FUNCTION_BLOCK FB_LensCompounderMock EXTENDS FB_FallibleMock IMPLEMENTS I_LensCompounder
VAR
    fFocalLengthCompounded : LREAL;
END_VAR


METHOD Compound : LREAL
VAR_INPUT
    fFocalLength	: LREAL;
    nMultiplier	: INT;
END_VAR
END_METHOD


PROPERTY FocalLengthCompounded : LREAL
GET

FocalLengthCompounded := fFocalLengthCompounded;
END_GET
SET

fFocalLengthCompounded := FocalLengthCompounded;
END_SET
END_PROPERTY


METHOD Reset
END_METHOD


METHOD SetValid

FocalLengthCompounded := 1.0;
ClearError();
END_METHOD

END_FUNCTION_BLOCK

(* stored: Version 1.1.0.1
   POU FB_LensCompounderMock: Id {f3a1ef28-98f7-4a8c-a126-ddef21ffe39c}, SpecialFunc None
   Method Compound: Id {785c0eab-8b59-435e-bd8e-fdfd5fe072fc}
   Property FocalLengthCompounded: Id {6ab06aab-6e17-48c9-8772-1a82ae1a3661}
   Get Get: Id {24dd4de6-a091-4797-9830-75cb541a3d9e}
   Set Set: Id {b9d8817e-a904-469f-93e9-2a1fa4393935}
   Method Reset: Id {899c1ae2-1f7c-43b4-bab3-4851756d6c8f}
   Method SetValid: Id {c1823eea-07dc-4ea6-ac07-5ee9857edefe} *)
